FUNCTION_BLOCK FB_CalcXRayDeltaElement_Test EXTENDS FB_TestSuiteExtended
VAR
    nTestID : INT;
END_VAR


nTestID := 0;

Test0AtomicMassExpectErrorDeltaUnchanged();

Test0AtomicNumberExpectErrorDeltaUnchanged();

Test0DensityExpectErrorDeltaUnchanged();

Test0EnergyExpectErrorDeltaUnchanged();

TestInvalidElementExpectErrorDeltaUnchanged();

TestInvalidEnergyExpectErrorDeltaUnchanged();

TestInvalidf1ExpectErrorDeltaUnchanged();

TestNegAtomicMassExpectErrorDeltaUnchanged();

TestNegAtomicNumberExpectErrorDeltaUnchanged();

TestNegDensityExpectErrorDeltaUnchanged();

TestNegEnergyExpectErrorDeltaUnchanged();

// Expected results taken from xraydb python module.
// Element = Be. Test Count = 1.
TestValidInputsExpectNoErrorAccurateDelta(
    fEnergy := 1000,
    fF1 := 0.12441385528833308,
    fDensity := 1.85,
    nAtomicNumber := 4,
    fAtomicMass := 9.0122,
    fExpected := 0.0003515107795702183
);

// Expected results taken from xraydb python module.
// Element = Be. Test Count = 2.
TestValidInputsExpectNoErrorAccurateDelta(
    fEnergy := 15000,
    fF1 := -0.00016936488385900804,
    fDensity := 1.85,
    nAtomicNumber := 4,
    fAtomicMass := 9.0122,
    fExpected := 1.515079754661661e-06
);

// Expected results taken from xraydb python module.
// Element = Be. Test Count = 3.
TestValidInputsExpectNoErrorAccurateDelta(
    fEnergy := 29000,
    fF1 := -0.0011666530513713296,
    fDensity := 1.85,
    nAtomicNumber := 4,
    fAtomicMass := 9.0122,
    fExpected := 4.052413187574221e-07
);

// Expected results taken from xraydb python module.
// Element = Ge. Test Count = 4.
TestValidInputsExpectNoErrorAccurateDelta(
    fEnergy := 1000,
    fF1 := -10.582299446346644,
    fDensity := 5.323,
    nAtomicNumber := 32,
    fAtomicMass := 72.63,
    fExpected := 0.0006517015706244444
);

// Expected results taken from xraydb python module.
// Element = Ge. Test Count = 5.
TestValidInputsExpectNoErrorAccurateDelta(
    fEnergy := 15000,
    fF1 := -0.20855631741810937,
    fDensity := 5.323,
    nAtomicNumber := 32,
    fAtomicMass := 72.63,
    fExpected := 4.299358473449007e-06
);

// Expected results taken from xraydb python module.
// Element = Ge. Test Count = 6.
TestValidInputsExpectNoErrorAccurateDelta(
    fEnergy := 29000,
    fF1 := 0.279006161044894,
    fDensity := 5.323,
    nAtomicNumber := 32,
    fAtomicMass := 72.63,
    fExpected := 1.1678850102602785e-06
);

// Expected results taken from xraydb python module.
// Element = C. Test Count = 7.
TestValidInputsExpectNoErrorAccurateDelta(
    fEnergy := 1000,
    fF1 := 0.32193839196465696,
    fDensity := 2.267,
    nAtomicNumber := 6,
    fAtomicMass := 12.011,
    fExpected := 0.0004954024109219588
);

// Expected results taken from xraydb python module.
// Element = C. Test Count = 8.
TestValidInputsExpectNoErrorAccurateDelta(
    fEnergy := 15000,
    fF1 := 0.003208693114407701,
    fDensity := 2.267,
    nAtomicNumber := 6,
    fAtomicMass := 12.011,
    fExpected := 2.0907821307300117e-06
);

// Expected results taken from xraydb python module.
// Element = C. Test Count = 9.
TestValidInputsExpectNoErrorAccurateDelta(
    fEnergy := 29000,
    fF1 := -0.0014327706311398664,
    fDensity := 2.267,
    nAtomicNumber := 6,
    fAtomicMass := 12.011,
    fExpected := 5.589325363478469e-07
);

// Expected results taken from xraydb python module.
// Element = Al. Test Count = 10.
TestValidInputsExpectNoErrorAccurateDelta(
    fEnergy := 1000,
    fF1 := -1.4706548748585362,
    fDensity := 2.7,
    nAtomicNumber := 13,
    fAtomicMass := 26.9815,
    fExpected := 0.000479002541009039
);

// Expected results taken from xraydb python module.
// Element = Al. Test Count = 11.
TestValidInputsExpectNoErrorAccurateDelta(
    fEnergy := 15000,
    fF1 := 0.08002784442214417,
    fDensity := 2.7,
    nAtomicNumber := 13,
    fAtomicMass := 26.9815,
    fExpected := 2.4152346347291635e-06
);

// Expected results taken from xraydb python module.
// Element = Al. Test Count = 12.
TestValidInputsExpectNoErrorAccurateDelta(
    fEnergy := 29000,
    fF1 := 0.01794721755836219,
    fDensity := 2.7,
    nAtomicNumber := 13,
    fAtomicMass := 26.9815,
    fExpected := 6.431017450275689e-07
);

// Expected results taken from xraydb python module.
// Element = Si. Test Count = 13.
TestValidInputsExpectNoErrorAccurateDelta(
    fEnergy := 1000,
    fF1 := -1.1466629849836463,
    fDensity := 2.329,
    nAtomicNumber := 14,
    fAtomicMass := 28.085,
    fExpected := 0.0004425338118167865
);

// Expected results taken from xraydb python module.
// Element = Si. Test Count = 14.
TestValidInputsExpectNoErrorAccurateDelta(
    fEnergy := 15000,
    fF1 := 0.10076225971581065,
    fDensity := 2.329,
    nAtomicNumber := 14,
    fAtomicMass := 28.085,
    fExpected := 2.1576978855198457e-06
);

// Expected results taken from xraydb python module.
// Element = Si. Test Count = 15.
TestValidInputsExpectNoErrorAccurateDelta(
    fEnergy := 29000,
    fF1 := 0.024412307252506597,
    fDensity := 2.329,
    nAtomicNumber := 14,
    fAtomicMass := 28.085,
    fExpected := 5.741418959262752e-07
);


METHOD PRIVATE SetInitialValues
VAR_IN_OUT
    fbQuantityLREALPublicEnergyMock : FB_QuantityLREALPublicMock;
    fbStringLookupLREALMock : FB_StringLookupLREALMock;
    fbStringLookupElementMock : FB_StringLookupElementMock;
END_VAR

fbQuantityLREALPublicEnergyMock.Val := 1.0;
fbQuantityLREALPublicEnergyMock.ClearError();

fbStringLookupLREALMock.Value := 1.0;
fbStringLookupLREALMock.ClearError();

fbStringLookupElementMock.Density := 1.0;
fbStringLookupElementMock.AtomicNumber := 1;
fbStringLookupElementMock.AtomicMass := 1.0;
fbStringLookupElementMock.ClearError();
END_METHOD


METHOD Test0AtomicMassExpectErrorDeltaUnchanged
VAR
    fbQuantityLREALPublicEnergyMock : FB_QuantityLREALPublicMock;
    fbStringLookupLREALMock : FB_StringLookupLREALMock;
    fbStringLookupElementMock : FB_StringLookupElementMock;
    fbExpected : FB_QuantityLREALPublicMock;
    fbConvertUnitsLREALMock : FB_ConvertUnitsLREALMock;

    // Subject under test
    fbCalcXRayDeltaElement : FB_CalcXRayDeltaElement(
        ConvertUnits := fbConvertUnitsLREALMock,
        Energy := fbQuantityLREALPublicEnergyMock,
        f1LUT := fbStringLookupLREALMock,
        ElementLUT := fbStringLookupElementMock
    );
    fbResult : FB_QuantityLREALPublic(Units := '1');
END_VAR

TEST('Test0AtomicMassExpectErrorDeltaUnchanged');

// Test fixture
SetInitialValues(
    fbQuantityLREALPublicEnergyMock := fbQuantityLREALPublicEnergyMock,
    fbStringLookupLREALMock := fbStringLookupLREALMock,
    fbStringLookupElementMock := fbStringLookupElementMock
);

fbStringLookupElementMock.AtomicMass := 0.0;

fbResult.Val := 5038.538;
fbExpected.Val := fbResult.Val;
fbExpected.Units := fbResult.Units;

// Here the test starts
fbCalcXRayDeltaElement.Calculate(
    MaterialFormula := 'Be',
    Delta := fbResult
);

AssertError(Fallible := fbCalcXRayDeltaElement);

AssertErrorExactExpectedQuantityLREAL(
    Expected := fbExpected,
    Actual := fbResult
);

TEST_FINISHED();
END_METHOD


METHOD Test0AtomicNumberExpectErrorDeltaUnchanged
VAR
    fbQuantityLREALPublicEnergyMock : FB_QuantityLREALPublicMock;
    fbStringLookupLREALMock : FB_StringLookupLREALMock;
    fbStringLookupElementMock : FB_StringLookupElementMock;
    fbExpected : FB_QuantityLREALPublicMock;
    fbConvertUnitsLREALMock : FB_ConvertUnitsLREALMock;

    // Subject under test
    fbCalcXRayDeltaElement : FB_CalcXRayDeltaElement(
        ConvertUnits := fbConvertUnitsLREALMock,
        Energy := fbQuantityLREALPublicEnergyMock,
        f1LUT := fbStringLookupLREALMock,
        ElementLUT := fbStringLookupElementMock
    );
    fbResult : FB_QuantityLREALPublic(Units := '1');
END_VAR

TEST('Test0AtomicNumberExpectErrorDeltaUnchanged');

// Test fixture
SetInitialValues(
    fbQuantityLREALPublicEnergyMock := fbQuantityLREALPublicEnergyMock,
    fbStringLookupLREALMock := fbStringLookupLREALMock,
    fbStringLookupElementMock := fbStringLookupElementMock
);

fbStringLookupElementMock.AtomicNumber := 0;

fbResult.Val := 5038.538;
fbExpected.Val := fbResult.Val;
fbExpected.Units := fbResult.Units;

// Here the test starts
fbCalcXRayDeltaElement.Calculate(
    MaterialFormula := 'Be',
    Delta := fbResult
);

AssertError(Fallible := fbCalcXRayDeltaElement);

AssertErrorExactExpectedQuantityLREAL(
    Expected := fbExpected,
    Actual := fbResult
);


TEST_FINISHED();
END_METHOD


METHOD Test0DensityExpectErrorDeltaUnchanged
VAR
    fbQuantityLREALPublicEnergyMock : FB_QuantityLREALPublicMock;
    fbStringLookupLREALMock : FB_StringLookupLREALMock;
    fbStringLookupElementMock : FB_StringLookupElementMock;
    fbExpected : FB_QuantityLREALPublicMock;
    fbConvertUnitsLREALMock : FB_ConvertUnitsLREALMock;

    // Subject under test
    fbCalcXRayDeltaElement : FB_CalcXRayDeltaElement(
        ConvertUnits := fbConvertUnitsLREALMock,
        Energy := fbQuantityLREALPublicEnergyMock,
        f1LUT := fbStringLookupLREALMock,
        ElementLUT := fbStringLookupElementMock
    );
    fbResult : FB_QuantityLREALPublic(Units := '1');
END_VAR

TEST('Test0DensityExpectErrorDeltaUnchanged');

// Test fixture
SetInitialValues(
    fbQuantityLREALPublicEnergyMock := fbQuantityLREALPublicEnergyMock,
    fbStringLookupLREALMock := fbStringLookupLREALMock,
    fbStringLookupElementMock := fbStringLookupElementMock
);

fbStringLookupElementMock.Density := 0.0;

fbResult.Val := 5038.538;
fbExpected.Val := fbResult.Val;
fbExpected.Units := fbResult.Units;

// Here the test starts
fbCalcXRayDeltaElement.Calculate(
    MaterialFormula := 'Be',
    Delta := fbResult
);

AssertError(Fallible := fbCalcXRayDeltaElement);

AssertErrorExactExpectedQuantityLREAL(
    Expected := fbExpected,
    Actual := fbResult
);

TEST_FINISHED();
END_METHOD


METHOD Test0EnergyExpectErrorDeltaUnchanged
VAR
    fbQuantityLREALPublicEnergyMock : FB_QuantityLREALPublicMock;
    fbStringLookupLREALMock : FB_StringLookupLREALMock;
    fbStringLookupElementMock : FB_StringLookupElementMock;
    fbExpected : FB_QuantityLREALPublicMock;
    fbConvertUnitsLREALMock : FB_ConvertUnitsLREALMock;

    // Subject under test
    fbCalcXRayDeltaElement : FB_CalcXRayDeltaElement(
        ConvertUnits := fbConvertUnitsLREALMock,
        Energy := fbQuantityLREALPublicEnergyMock,
        f1LUT := fbStringLookupLREALMock,
        ElementLUT := fbStringLookupElementMock
    );
    fbResult : FB_QuantityLREALPublic(Units := '1');
END_VAR

TEST('Test0EnergyExpectErrorDeltaUnchanged');

// Test fixture
SetInitialValues(
    fbQuantityLREALPublicEnergyMock := fbQuantityLREALPublicEnergyMock,
    fbStringLookupLREALMock := fbStringLookupLREALMock,
    fbStringLookupElementMock := fbStringLookupElementMock
);

fbQuantityLREALPublicEnergyMock.Val := 0.0;

fbResult.Val := 5038.538;
fbExpected.Val := fbResult.Val;
fbExpected.Units := fbResult.Units;

// Here the test starts
fbCalcXRayDeltaElement.Calculate(
    MaterialFormula := 'Be',
    Delta := fbResult
);

AssertError(Fallible := fbCalcXRayDeltaElement);

AssertErrorExactExpectedQuantityLREAL(
    Expected := fbExpected,
    Actual := fbResult
);

TEST_FINISHED();
END_METHOD


METHOD TestInvalidElementExpectErrorDeltaUnchanged
VAR
    fbQuantityLREALPublicEnergyMock : FB_QuantityLREALPublicMock;
    fbStringLookupLREALMock : FB_StringLookupLREALMock;
    fbStringLookupElementMock : FB_StringLookupElementMock;
    fbExpected : FB_QuantityLREALPublicMock;
    fbConvertUnitsLREALMock : FB_ConvertUnitsLREALMock;

    // Subject under test
    fbCalcXRayDeltaElement : FB_CalcXRayDeltaElement(
        ConvertUnits := fbConvertUnitsLREALMock,
        Energy := fbQuantityLREALPublicEnergyMock,
        f1LUT := fbStringLookupLREALMock,
        ElementLUT := fbStringLookupElementMock
    );
    fbResult : FB_QuantityLREALPublic(Units := '1');
END_VAR

TEST('TestInvalidElementExpectErrorDeltaUnchanged');

// Test fixture
SetInitialValues(
    fbQuantityLREALPublicEnergyMock := fbQuantityLREALPublicEnergyMock,
    fbStringLookupLREALMock := fbStringLookupLREALMock,
    fbStringLookupElementMock := fbStringLookupElementMock
);

fbStringLookupElementMock.SetError(Msg := 'Error');

fbResult.Val := 5038.538;
fbExpected.Val := fbResult.Val;
fbExpected.Units := fbResult.Units;

// Here the test starts
fbCalcXRayDeltaElement.Calculate(
    MaterialFormula := 'Be',
    Delta := fbResult
);

AssertError(Fallible := fbCalcXRayDeltaElement);

AssertErrorExactExpectedQuantityLREAL(
    Expected := fbExpected,
    Actual := fbResult
);

TEST_FINISHED();
END_METHOD


METHOD TestInvalidEnergyExpectErrorDeltaUnchanged
VAR
    fbQuantityLREALPublicEnergyMock : FB_QuantityLREALPublicMock;
    fbStringLookupLREALMock : FB_StringLookupLREALMock;
    fbStringLookupElementMock : FB_StringLookupElementMock;
    fbExpected : FB_QuantityLREALPublicMock;
    fbConvertUnitsLREALMock : FB_ConvertUnitsLREALMock;

    // Subject under test
    fbCalcXRayDeltaElement : FB_CalcXRayDeltaElement(
        ConvertUnits := fbConvertUnitsLREALMock,
        Energy := fbQuantityLREALPublicEnergyMock,
        f1LUT := fbStringLookupLREALMock,
        ElementLUT := fbStringLookupElementMock
    );
    fbResult : FB_QuantityLREALPublic(Units := '1');
END_VAR

TEST('TestInvalidEnergyExpectErrorDeltaUnchanged');

// Test fixture
SetInitialValues(
    fbQuantityLREALPublicEnergyMock := fbQuantityLREALPublicEnergyMock,
    fbStringLookupLREALMock := fbStringLookupLREALMock,
    fbStringLookupElementMock := fbStringLookupElementMock
);

fbQuantityLREALPublicEnergyMock.SetError(Msg := 'Error');

fbResult.Val := 5038.538;
fbExpected.Val := fbResult.Val;
fbExpected.Units := fbResult.Units;

// Here the test starts
fbCalcXRayDeltaElement.Calculate(
    MaterialFormula := 'Be',
    Delta := fbResult
);

AssertError(Fallible := fbCalcXRayDeltaElement);

AssertErrorExactExpectedQuantityLREAL(
    Expected := fbExpected,
    Actual := fbResult
);
TEST_FINISHED();
END_METHOD


METHOD TestInvalidf1ExpectErrorDeltaUnchanged
VAR
    fbQuantityLREALPublicEnergyMock : FB_QuantityLREALPublicMock;
    fbStringLookupLREALMock : FB_StringLookupLREALMock;
    fbStringLookupElementMock : FB_StringLookupElementMock;
    fbExpected : FB_QuantityLREALPublicMock;
    fbConvertUnitsLREALMock : FB_ConvertUnitsLREALMock;

    // Subject under test
    fbCalcXRayDeltaElement : FB_CalcXRayDeltaElement(
        ConvertUnits := fbConvertUnitsLREALMock,
        Energy := fbQuantityLREALPublicEnergyMock,
        f1LUT := fbStringLookupLREALMock,
        ElementLUT := fbStringLookupElementMock
    );
    fbResult : FB_QuantityLREALPublic(Units := '1');
END_VAR

TEST('TestInvalidf1ExpectErrorDeltaUnchanged');

// Test fixture
SetInitialValues(
    fbQuantityLREALPublicEnergyMock := fbQuantityLREALPublicEnergyMock,
    fbStringLookupLREALMock := fbStringLookupLREALMock,
    fbStringLookupElementMock := fbStringLookupElementMock
);

fbStringLookupLREALMock.SetError(Msg := 'Error');

fbResult.Val := 5038.538;
fbExpected.Val := fbResult.Val;
fbExpected.Units := fbResult.Units;

// Here the test starts
fbCalcXRayDeltaElement.Calculate(
    MaterialFormula := 'Be',
    Delta := fbResult
);

AssertError(Fallible := fbCalcXRayDeltaElement);

AssertErrorExactExpectedQuantityLREAL(
    Expected := fbExpected,
    Actual := fbResult
);

TEST_FINISHED();
END_METHOD


METHOD TestNegAtomicMassExpectErrorDeltaUnchanged
VAR
    fbQuantityLREALPublicEnergyMock : FB_QuantityLREALPublicMock;
    fbStringLookupLREALMock : FB_StringLookupLREALMock;
    fbStringLookupElementMock : FB_StringLookupElementMock;
    fbExpected : FB_QuantityLREALPublicMock;
    fbConvertUnitsLREALMock : FB_ConvertUnitsLREALMock;

    // Subject under test
    fbCalcXRayDeltaElement : FB_CalcXRayDeltaElement(
        ConvertUnits := fbConvertUnitsLREALMock,
        Energy := fbQuantityLREALPublicEnergyMock,
        f1LUT := fbStringLookupLREALMock,
        ElementLUT := fbStringLookupElementMock
    );
    fbResult : FB_QuantityLREALPublic(Units := '1');
END_VAR

TEST('TestNegAtomicMassExpectErrorDeltaUnchanged');

// Test fixture
SetInitialValues(
    fbQuantityLREALPublicEnergyMock := fbQuantityLREALPublicEnergyMock,
    fbStringLookupLREALMock := fbStringLookupLREALMock,
    fbStringLookupElementMock := fbStringLookupElementMock
);

fbStringLookupElementMock.AtomicMass := -10.0;

fbResult.Val := 5038.538;
fbExpected.Val := fbResult.Val;
fbExpected.Units := fbResult.Units;

// Here the test starts
fbCalcXRayDeltaElement.Calculate(
    MaterialFormula := 'Be',
    Delta := fbResult
);

AssertError(Fallible := fbCalcXRayDeltaElement);

AssertErrorExactExpectedQuantityLREAL(
    Expected := fbExpected,
    Actual := fbResult
);

TEST_FINISHED();
END_METHOD


METHOD TestNegAtomicNumberExpectErrorDeltaUnchanged
VAR
    fbQuantityLREALPublicEnergyMock : FB_QuantityLREALPublicMock;
    fbStringLookupLREALMock : FB_StringLookupLREALMock;
    fbStringLookupElementMock : FB_StringLookupElementMock;
    fbExpected : FB_QuantityLREALPublicMock;
    fbConvertUnitsLREALMock : FB_ConvertUnitsLREALMock;

    // Subject under test
    fbCalcXRayDeltaElement : FB_CalcXRayDeltaElement(
        ConvertUnits := fbConvertUnitsLREALMock,
        Energy := fbQuantityLREALPublicEnergyMock,
        f1LUT := fbStringLookupLREALMock,
        ElementLUT := fbStringLookupElementMock
    );
    fbResult : FB_QuantityLREALPublic(Units := '1');
END_VAR

TEST('TestNegAtomicNumberExpectErrorDeltaUnchanged');

// Test fixture
SetInitialValues(
    fbQuantityLREALPublicEnergyMock := fbQuantityLREALPublicEnergyMock,
    fbStringLookupLREALMock := fbStringLookupLREALMock,
    fbStringLookupElementMock := fbStringLookupElementMock
);

fbStringLookupElementMock.AtomicNumber := -10;

fbResult.Val := 5038.538;
fbExpected.Val := fbResult.Val;
fbExpected.Units := fbResult.Units;

// Here the test starts
fbCalcXRayDeltaElement.Calculate(
    MaterialFormula := 'Be',
    Delta := fbResult
);

AssertError(Fallible := fbCalcXRayDeltaElement);

AssertErrorExactExpectedQuantityLREAL(
    Expected := fbExpected,
    Actual := fbResult
);

TEST_FINISHED();
END_METHOD


METHOD TestNegDensityExpectErrorDeltaUnchanged
VAR
    fbQuantityLREALPublicEnergyMock : FB_QuantityLREALPublicMock;
    fbStringLookupLREALMock : FB_StringLookupLREALMock;
    fbStringLookupElementMock : FB_StringLookupElementMock;
    fbExpected : FB_QuantityLREALPublicMock;
    fbConvertUnitsLREALMock : FB_ConvertUnitsLREALMock;

    // Subject under test
    fbCalcXRayDeltaElement : FB_CalcXRayDeltaElement(
        ConvertUnits := fbConvertUnitsLREALMock,
        Energy := fbQuantityLREALPublicEnergyMock,
        f1LUT := fbStringLookupLREALMock,
        ElementLUT := fbStringLookupElementMock
    );
    fbResult : FB_QuantityLREALPublic(Units := '1');
END_VAR

TEST('TestNegDensityExpectErrorDeltaUnchanged');

// Test fixture
SetInitialValues(
    fbQuantityLREALPublicEnergyMock := fbQuantityLREALPublicEnergyMock,
    fbStringLookupLREALMock := fbStringLookupLREALMock,
    fbStringLookupElementMock := fbStringLookupElementMock
);

fbStringLookupElementMock.Density := 0.0;

fbResult.Val := 5038.538;
fbExpected.Val := fbResult.Val;
fbExpected.Units := fbResult.Units;

// Here the test starts
fbCalcXRayDeltaElement.Calculate(
    MaterialFormula := 'Be',
    Delta := fbResult
);

AssertError(Fallible := fbCalcXRayDeltaElement);

AssertErrorExactExpectedQuantityLREAL(
    Expected := fbExpected,
    Actual := fbResult
);

TEST_FINISHED();
END_METHOD


METHOD TestNegEnergyExpectErrorDeltaUnchanged
VAR
    fbQuantityLREALPublicEnergyMock : FB_QuantityLREALPublicMock;
    fbStringLookupLREALMock : FB_StringLookupLREALMock;
    fbStringLookupElementMock : FB_StringLookupElementMock;
    fbExpected : FB_QuantityLREALPublicMock;
    fbConvertUnitsLREALMock : FB_ConvertUnitsLREALMock;

    // Subject under test
    fbCalcXRayDeltaElement : FB_CalcXRayDeltaElement(
        ConvertUnits := fbConvertUnitsLREALMock,
        Energy := fbQuantityLREALPublicEnergyMock,
        f1LUT := fbStringLookupLREALMock,
        ElementLUT := fbStringLookupElementMock
    );
    fbResult : FB_QuantityLREALPublic(Units := '1');
END_VAR

TEST('TestNegEnergyExpectErrorDeltaUnchanged');

// Test fixture
SetInitialValues(
    fbQuantityLREALPublicEnergyMock := fbQuantityLREALPublicEnergyMock,
    fbStringLookupLREALMock := fbStringLookupLREALMock,
    fbStringLookupElementMock := fbStringLookupElementMock
);

fbQuantityLREALPublicEnergyMock.Val := 0.0;

fbResult.Val := 5038.538;
fbExpected.Val := fbResult.Val;
fbExpected.Units := fbResult.Units;

// Here the test starts
fbCalcXRayDeltaElement.Calculate(
    MaterialFormula := 'Be',
    Delta := fbResult
);

AssertError(Fallible := fbCalcXRayDeltaElement);

AssertErrorExactExpectedQuantityLREAL(
    Expected := fbExpected,
    Actual := fbResult
);

TEST_FINISHED();
END_METHOD


METHOD TestValidInputsExpectNoErrorAccurateDelta
VAR_INPUT
    fEnergy : LREAL;
    fF1 : LREAL;
    fDensity : LREAL;
    nAtomicNumber : INT;
    fAtomicMass : LREAL;

    fExpected : LREAL;
END_VAR
VAR
    fbQuantityLREALPublicEnergyMock : FB_QuantityLREALPublicMock;
    fbStringLookupLREALMock : FB_StringLookupLREALMock;
    fbStringLookupElementMock : FB_StringLookupElementMock;
    fbExpected : FB_QuantityLREALPublicMock;
    fbConvertUnitsLREALMock : FB_ConvertUnitsLREALMock;

    // Subject under test
    fbCalcXRayDeltaElement : FB_CalcXRayDeltaElement(
        ConvertUnits := fbConvertUnitsLREALMock,
        Energy := fbQuantityLREALPublicEnergyMock,
        f1LUT := fbStringLookupLREALMock,
        ElementLUT := fbStringLookupElementMock
    );
    fbResult : FB_QuantityLREALPublic(Units := '1');
END_VAR

TEST(CONCAT(STR1 := 'TestValidInputsExpectNoErrorAccurateDelta ID: ',
            STR2 := INT_TO_STRING(nTestID)));

// Test fixture
SetInitialValues(
    fbQuantityLREALPublicEnergyMock := fbQuantityLREALPublicEnergyMock,
    fbStringLookupLREALMock := fbStringLookupLREALMock,
    fbStringLookupElementMock := fbStringLookupElementMock
);

fbQuantityLREALPublicEnergyMock.Val := fEnergy;
fbStringLookupLREALMock.Value := fF1;
fbStringLookupElementMock.Density := fDensity;
fbStringLookupElementMock.AtomicNumber := nAtomicNumber;
fbStringLookupElementMock.AtomicMass := fAtomicMass;

fbExpected.Val := fExpected;
fbExpected.Units := fbResult.Units;

// Here the test starts
fbCalcXRayDeltaElement.Calculate(
    MaterialFormula := 'Be',
    Delta := fbResult
);

AssertNoError(Fallible := fbCalcXRayDeltaElement);

AssertNoErrorExpectedQuantityLREAL(
    Expected := fbExpected,
    Actual := fbResult,
    Delta := ABS(0.001 * fbExpected.Val)
);

TEST_FINISHED();

nTestID := nTestID + 1;
END_METHOD

END_FUNCTION_BLOCK

(* stored: Version 1.1.0.1
   POU FB_CalcXRayDeltaElement_Test: Id {98858369-0487-4f19-ba02-1eea298ccad3}, SpecialFunc None
   Method SetInitialValues: Id {f04845fb-8191-4651-bfc2-72b1efacd442}
   Method Test0AtomicMassExpectErrorDeltaUnchanged: Id {b6dc767c-cf65-41d6-8be0-32b5df8d14ad}
   Method Test0AtomicNumberExpectErrorDeltaUnchanged: Id {19f8aed2-3809-4397-9ebb-60e03b7208cf}
   Method Test0DensityExpectErrorDeltaUnchanged: Id {a22c9ec5-6265-4c4b-81b1-88d5546cb3c5}
   Method Test0EnergyExpectErrorDeltaUnchanged: Id {27c084a3-dc63-4167-a57f-ff90d70c622f}
   Method TestInvalidElementExpectErrorDeltaUnchanged: Id {6e484356-c61f-45c5-80a8-578577b9fc57}
   Method TestInvalidEnergyExpectErrorDeltaUnchanged: Id {708d60b9-322c-4b04-ac4c-a6f261d3e002}
   Method TestInvalidf1ExpectErrorDeltaUnchanged: Id {0fc9efb7-0fe3-4d4f-9e8d-8ecac8e37e76}
   Method TestNegAtomicMassExpectErrorDeltaUnchanged: Id {1fe53040-1c34-4a85-99a3-d4bfb0bd91fb}
   Method TestNegAtomicNumberExpectErrorDeltaUnchanged: Id {da7f21be-bbb5-4949-8587-a784e59a2f1d}
   Method TestNegDensityExpectErrorDeltaUnchanged: Id {7770c05a-bc0a-490d-8217-61adc2d656a7}
   Method TestNegEnergyExpectErrorDeltaUnchanged: Id {74f08a4b-e970-41a6-8f17-caa755927812}
   Method TestValidInputsExpectNoErrorAccurateDelta: Id {98dcca39-02f5-4794-8d0d-043b48f5e73a} *)
